PROGRAM AlarmExtension
VAR
	bAlarm		: BOOL;
	iAlarm		: INT;
END_VAR

END_PROGRAM

(* stored: Version 1.1.0.1, ProductVersion 3.1.4024.12
   POU AlarmExtension: Id {7495b61b-c2b8-43af-8049-87b29744281f}, SpecialFunc None *)
